(* CODESYS project Azure_IOTDevicePi_RECOVERED_2025-06-12T00-39-57.project

Project tree, tasks and I/O mapping:
  Device : CODESYS Control for Raspberry Pi SL, CODESYS, order no. 2302000009, version 4.12.0.0
    application Application
      libraries: Standard, 3.5.18.0 (System); Azure IoT Hub Client SL, 1.9.0.0 (CODESYS); StringUtils, 3.5.20.0 (System); SysTimeRtc, * (System); CAA Net Base Services, * (CAA Technical Workgroup); VisuDialogs, * (System)
      task MainTask (freewheeling, priority 1) calls MQTT_Comms, Sockets_Server, RobotPP
      task VISU_TASK (cyclic, interval 100 ms, priority 31) calls VisuElems.Visu_Prg
      HMI/
        Tags/
          global variables HMI_GV
        Visu/
          visualisation Home
        UDTs/
          data type HMI_UDT
      PLC/
        UDTs/
        Logic/
          program RobotPP [LD]
          program Sockets_Server [ST]
          program MQTT_Comms [ST]: Build_Send_Message
        Tags/
    I²C
    Camera device
      <Empty>
    SPI
    GPIOs_A_B : GPIOs A/B, CODESYS, version 4.12.0.0
        unmapped channels: digital inputs (GPIO0..GPIO31), digital outputs (GPIO0..GPIO31)
    SoftMotion General Axis Pool
    Onewire
  5ce3da45-db07-42e7-a21c-a00fff4ed8f6|C:\Temp\background.jpg
  image pool ImagePool
  text list ConnectedStatus
  text list GlobalTextList
*)

// Device/Application/HMI/UDTs/HMI_UDT
TYPE HMI_UDT :
STRUCT
	CYCLE_START_PB: BOOL;
	CYCLE_STOP_PB: BOOL;
	ENABLE_TCP_SRV_PB:BOOL;
	TIME_SS: DINT;
	TIME_MIN:DINT;
	TIME_HH:DINT;
	TIME_YYYY:DINT;
	TIME_MM:DINT;
	TIME_DD:DINT;
	
END_STRUCT
END_TYPE

// Device/Application/HMI/Tags/HMI_GV
{attribute 'qualified_only'}
VAR_GLOBAL PERSISTENT RETAIN
	HMI: HMI_UDT;
END_VAR

// Device/Application/PLC/Logic/MQTT_Comms
PROGRAM MQTT_Comms
VAR
	sSubDomainName : STRING(100) := 'lrIOT'; // The name Azure IoT Hub
	sDeviceId : STRING(100) := 'myDevice01'; // The device id
	wsDeviceSaS : WSTRING(255) := "SharedAccessSignature sr=lrIOT.azure-devices.net%2Fdevices%2FmyDevice01&sig=TaqGGGcvZcrZOEFWE4%2Fymzi%2F2j20MA0J4v39ltraJkY%3D&se=1749931581"; // Your device SaS token (needed for c2d and d2c messages)

	azureMqttClient : AZURE.AzureMQTTClient; // Function block to establish a MQTT connection to Azure IoT Hub
	xConnect : BOOL; // TRUE: Connect to IoT Hub
	sendMQTTMessage : AZURE.SendMQTTMessage; // Function block to send a D2C message via MQTT to Azure IoT Hub
	
	sSendMessage : STRING(4095); // D2C message (send)
	
END_VAR

//MQTT Comms - Functions Instances

//Built String to Send to   Azure
sSendMessage:= 	MQTT_Comms.Build_Send_Message();

// Create a connection via MQTT
azureMqttClient(	xEnable := RobotPP.RobotInCycle,
					uiKeepAlive := 10,
					sHubDomainName := sSubDomainName,
					sDeviceId := sDeviceId,
					wsSaS := wsDeviceSaS);
					
					
// Send D2C messages						
sendMQTTMessage( 	xExecute := RobotPP.Write_MQTT_Msg,
					udiTimeOut := 2000000,
					pbPayload := ADR(sSendMessage),
					udiPayloadSize := DINT_TO_UDINT(Stu.StrLenA(ADR(sSendMessage))),
					azureMQTTClient := azureMqttClient);

METHOD Build_Send_Message : STRING(4095)
VAR_INPUT
END_VAR

VAR
	str_build: STRING(4095);
	Date_and_time_in_seconds : UDINT;
	Local_date_time_seconds : UDINT;
	Date_and_Time_result : UDINT;
	Date_and_time_format : DATE_AND_TIME;
	Date_and_time_string : STRING;
END_VAR

// Get time in seconds since 1970 :
Date_and_time_in_seconds := SysTimeRtcGet(Date_and_Time_result);
IF Date_and_Time_result <> 0 THEN
RETURN;
END_IF

// Convert UTC seconds to local time seconds, regarding Timezone and Summer time :
Date_and_Time_result := SysTimeRtcConvertUtcToLocal(Date_and_time_in_seconds, Local_date_time_seconds);
IF Date_and_Time_result <> 0 THEN
RETURN;
END_IF

// Convert the local seconds to a DATE_AND_TIME variable dt#yyyy-mm-dd-hh:mm:ss :
Date_and_time_format := UDINT_TO_DT(Local_date_time_seconds);

// Convert DATE_AND_TIME to a String :
Date_and_time_string := DT_TO_STRING(Date_and_time_format);

HMI_GV.HMI.TIME_YYYY := STRING_TO_INT(Mid(date_and_time_string, 4, 4));
HMI_GV.HMI.TIME_MM := STRING_TO_INT(Mid(date_and_time_string, 2, 9));
HMI_GV.HMI.TIME_DD := STRING_TO_INT(Mid(date_and_time_string, 2, 12));
HMI_GV.HMI.TIME_HH := STRING_TO_INT(Mid(date_and_time_string, 2, 15));
HMI_GV.HMI.TIME_MIN := STRING_TO_INT(MID(date_and_time_string, 2, 18));
HMI_GV.HMI.TIME_SS := STRING_TO_INT(right(date_and_time_string,2));



//str_build:= CONCAT('{ $"messageId$" :', '');
str_build:= CONCAT('{ $"ProdCount$" :', DINT_TO_STRING(Sockets_Server.ReadData[1]));
str_build:= CONCAT(str_build, ', $"deviceId$" : $"CodesysRobotPP$", ');
//str_build:= CONCAT(str_build, '$"temperature$" : 26, ');
//str_build:= CONCAT(str_build, '$"humidity$" : 32, ');
str_build:= CONCAT(str_build, '$"timestamp$" : "');
str_build:= CONCAT(str_build, RIGHT(Date_and_time_string,19));
str_build:= CONCAT(str_build, '"}');

Build_Send_Message:= str_build;
END_METHOD

END_PROGRAM

// Device/Application/PLC/Logic/RobotPP
PROGRAM RobotPP
VAR
	Cycle_Start: BOOL;
	Cycle_Complete: BOOL;
	RobotInCycle: BOOL;
	R_TRIG_0: R_TRIG;
	Write_MQTT_Msg: BOOL;
END_VAR
VAR // added by the converter: edge detectors and wires of the graphical bodies
    _w1, _w2, _w3 : BOOL;
END_VAR

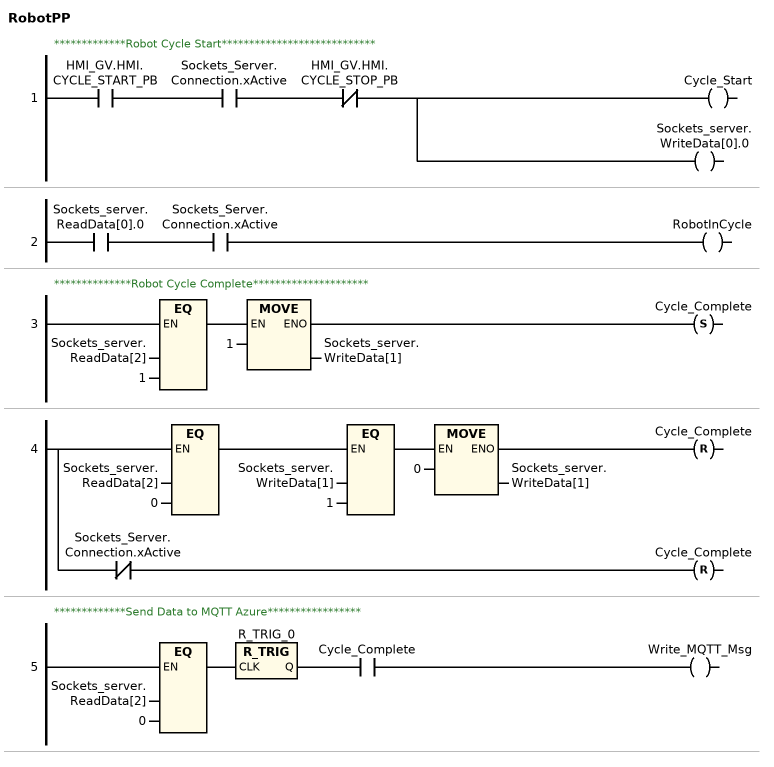
// NETWORK 1
// *************Robot Cycle Start****************************
_w1 := HMI_GV.HMI.CYCLE_START_PB AND Sockets_Server.Connection.xActive AND NOT HMI_GV.HMI.CYCLE_STOP_PB;
Cycle_Start := _w1;
Sockets_server.WriteData[0].0 := _w1;

// NETWORK 2
RobotInCycle := Sockets_server.ReadData[0].0 AND Sockets_Server.Connection.xActive;

// NETWORK 3
// **************Robot Cycle Complete*********************
_w2 := Sockets_server.ReadData[2] = 1;
IF _w2 THEN Sockets_server.WriteData[1] := 1; END_IF
Cycle_Complete S= _w2;

// NETWORK 4
_w3 := Sockets_server.ReadData[2] = 0 AND Sockets_server.WriteData[1] = 1;
IF _w3 THEN Sockets_server.WriteData[1] := 0; END_IF
Cycle_Complete R= _w3;
Cycle_Complete R= NOT Sockets_Server.Connection.xActive;

// NETWORK 5
// *************Send Data to MQTT Azure*****************
R_TRIG_0(CLK := Sockets_server.ReadData[2] = 0); // R_TRIG
Write_MQTT_Msg := R_TRIG_0.Q AND Cycle_Complete;

END_PROGRAM

// Device/Application/PLC/Logic/Sockets_Server
PROGRAM Sockets_Server
VAR
    ipAddr : NBS.IP_ADDR := (sAddr:='25.38.171.74');
	Server: NBS.TCP_Server :=(uiPort :=49151);
	

	Connection: NBS.TCP_Connection;
	Read : NBS.TCP_Read;
	Write : NBS.TCP_Write;
	
	T1: TON := (PT := TIME#50MS);
	xEnableServer: BOOL;
	
	ReadData: ARRAY[0..3] OF DINT;
END_VAR
VAR_INPUT
	WriteData:  ARRAY[0..3] OF DINT;
END_VAR

//TCP Sockets Server

//Server Instance
Server(xEnable:=HMI_GV.HMI.ENABLE_TCP_SRV_PB,
		ipAddr:= ipAddr
		);
		
//Conection INstance	
Connection(xEnable:=(Server.xbusy AND NOT(Connection.xDone)),
		hServer:= Server.hServer
		);
		
//Read Data		
Read(xEnable:= Connection.xActive,
		hConnection:=Connection.hConnection,
		szSize:=SIZEOF(ReadData),
		pData:=ADR(ReadData)
		);
		
//Write Data	
Write(xExecute:= Connection.xActive AND T1.Q,
		hConnection:=Connection.hConnection,
		szSize:=SIZEOF(WriteData),
		pData:=ADR(WriteData)
		);

//Write Data Time Interval	
T1(IN:=NOT(Write.xDone));

END_PROGRAM

// Device/Application/HMI/Visu/Home
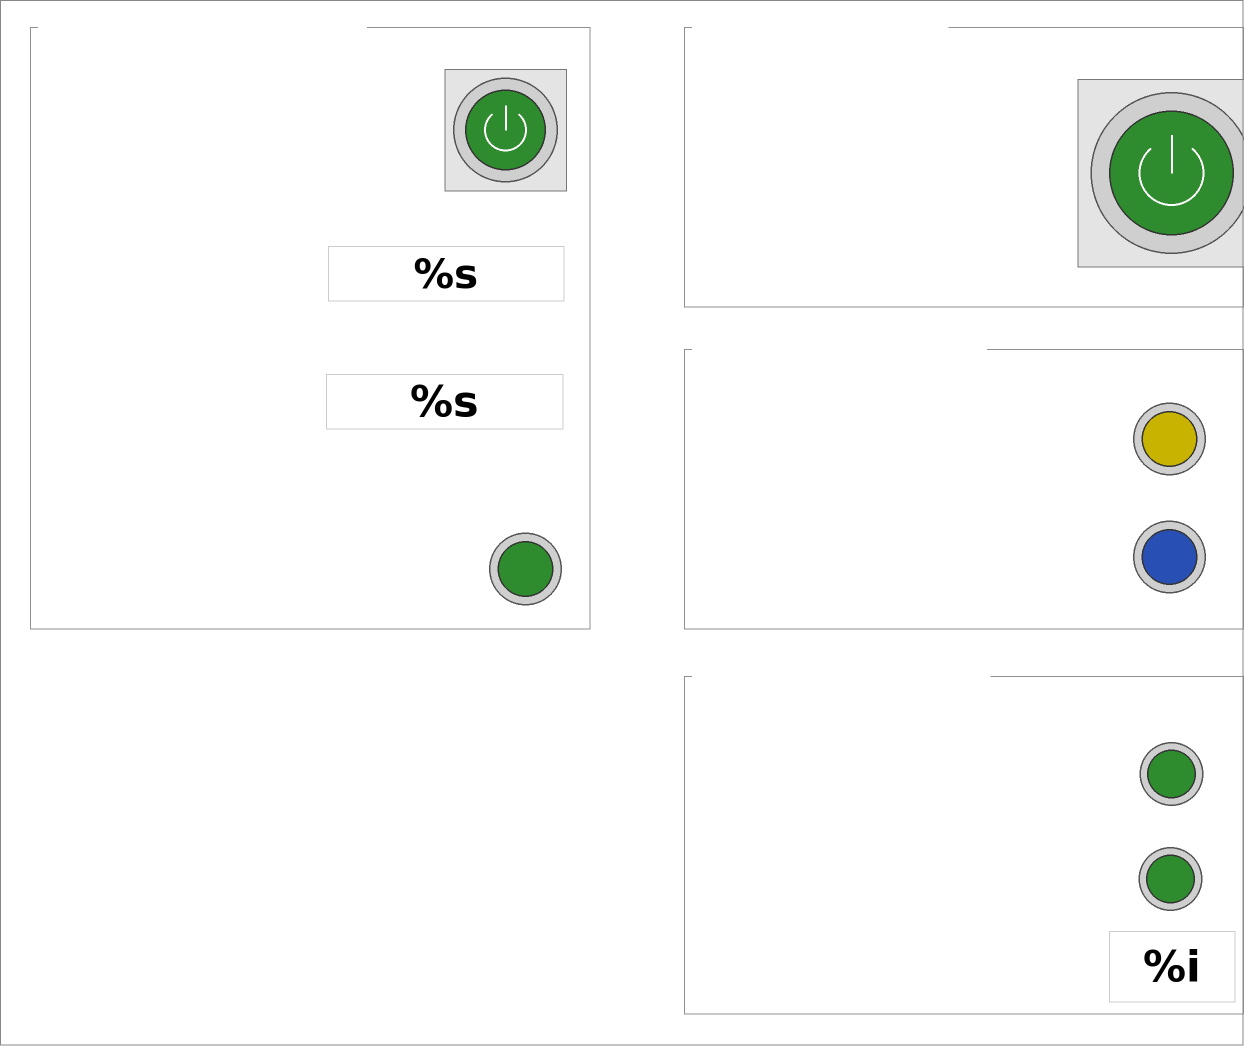
VISUALIZATION Home  // 1244x1046, background image ImagePool.background
    GroupBox (684,19 560x288), "Cycle Start"
        PowerSwitch (346,60 283x188), tooltip "Connect", variable: HMI_GV.HMI.CYCLE_START_PB, behaviour: TOGGLE, style: Switch-PowerSwitch-Green
    GroupBox (684,341 560x288), "MQTT Status"
        Lamp1 (437,56 97x84), variable: MQTT_Comms.azureMqttClient.xConnectedToBroker, style: Lamp-Lamp1-Yellow
        Label (116,57 203x73), "Connected"
        Label (116,165 250x73), "Data Uploaded"
        Lamp1 (437,174 97x84), variable: MQTT_Comms.sendMQTTMessage.xDone, style: Lamp-Lamp1-Blue
    GroupBox (684,668 560x346), "Robot Status"
        Label (116,57 203x73), "In Cycle"
        Label (116,165 250x73), "Cycle Completed"
        Lamp1 (441,69 93x74), variable: RobotPP.RobotInCycle, style: Lamp-Lamp1-Green
        Lamp1 (440,174 93x74), variable: Sockets_Server.ReadData[2].0, style: Lamp-Lamp1-Green
    Textfield (1109,931 126x71), "%i", text variable: Sockets_Server.ReadData[1]
    Label (800,910 285x136), "Completed Cycles Count"
    GroupBox (30,19 560x610), "Sockets Server"
        Label (22,84 249x69), "Enable Server"
        Lamp1 (447,508 97x84), variable: Sockets_Server.Connection.xActive, style: Lamp-Lamp1-Green
        Textfield (298,227 236x55), "%s", text variable: Sockets_Server.ipAddr.sAddr
            OnMouseClick: write the text variable via VisuDialogs.Numpad
        Label (22,219 336x73), "Server Address"
        PowerSwitch (407,50 137x122), tooltip "Connect", variable: HMI_GV.HMI.ENABLE_TCP_SRV_PB, behaviour: TOGGLE, style: Switch-PowerSwitch-Green
        Textfield (296,355 237x55), "%s", text variable: Sockets_Server.Server.uiPort
            OnMouseClick: write the text variable via VisuDialogs.Numpad
        Textfield (22,525 507x55), "%s", text list: 'ConnectedStatus', text index: Sockets_Server.Connection.xActive
            OnMouseClick: write the text variable via VisuDialogs.Numpad
        Label (22,337 336x73), "Server Port"
END_VISUALIZATION

(* text list ConnectedStatus (id | default)
  0 | Waiting Client Connection
  1 | Client Connected
   |  *)
